ABB RobotStudio station: 2. undervisning_20200306-072351.rsstn

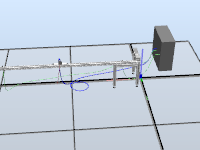
Station 2. undervisning (saved by RobotStudio 7.0.8728.594)
Layout (positions relative to the parent item):
  - base_2 [part] at (0, 0, -80) mm, rotated rx 90 ry 0 rz 0 deg
  - cart_2 [part] at (735.31, -25, 445) mm, rotated rx 90 ry 0 rz 0 deg
  - Part_3 [part]
  - pendul [part] at (1135.31, 239.5, 479.97) mm, rotated rx 90 ry -9.41 rz 0 deg
  - Part_8 [part] at (0, 0, 0) mm
  - Part_9 [part] at (0, 0, 0) mm
  - Part_10 [part]
  - PhysicsCable_1 [physicscable]
  - Part_13 [part]
  - Part_14 [part]
  - PhysicsCable_4 [physicscable]
  - PhysicsCable_5 [physicscable]
